Fanuc KAREL source: kt00518.KL

-- PROVISIONAL review KL for V940-1; original PC SHA256 7ce1e686dda61532a97a6188272de02c0082f0f1f3c53049c5b8473b59b4f1c3
-- Incomplete behavior may be omitted. Consult companion uncertainty JSON. Do not deploy.
PROGRAM KT00518
%NOLOCKGROUP
VAR
  OUT : BOOLEAN
-- UNRESOLVED_DECL P1 type=000106
-- UNRESOLVED_DECL P2 type=000102
BEGIN
  -- V9_ZERO_TABLE_METADATA_HINT layout=0001; no indexed target words; source/name/runtime held
  -- UNRESOLVED_PC offsets 5-20; opcodes 2E,22,32,35
  -- UNRESOLVED_PC offsets 25-40; opcodes 2E,22,32,35
  -- UNRESOLVED_PC offsets 45-78; opcodes 49,7E,49,7E,AC,23
  -- UNRESOLVED_PC offsets 83-87; opcodes 7F
END KT00518
